// Mitsubishi GX Works2 project: modbus ASCII   PLC: FX1N/FX1NC

PROGRAM MAIN
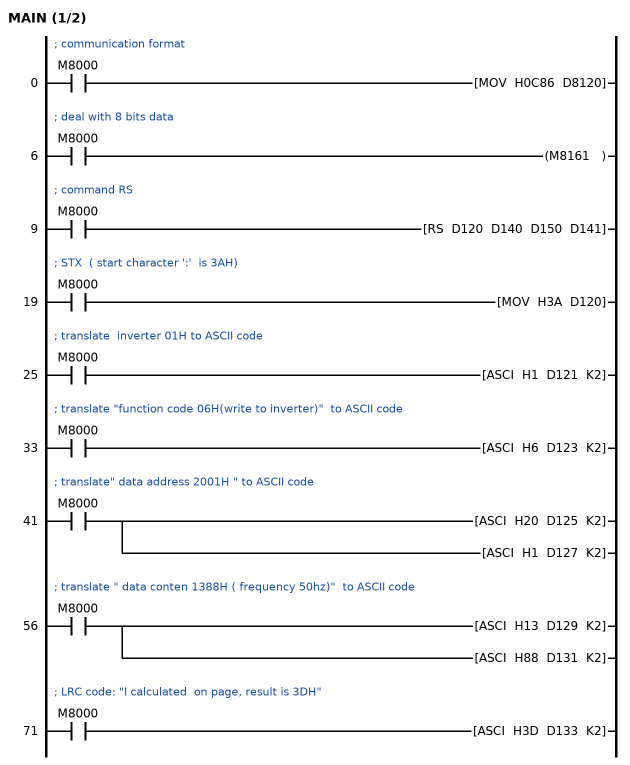
; communication format
0     LD      M8000
      MOV     H0C86 D8120
; deal with 8 bits data
6     LD      M8000
      OUT     M8161
; command RS
9     LD      M8000
      RS      D120 D140 D150 D141
; STX  ( start character ':'  is 3AH)
19    LD      M8000
      MOV     H3A D120
; translate  inverter 01H to ASCII code
25    LD      M8000
      ASCI    H1 D121 K2
; translate "function code 06H(write to inverter)"  to ASCII code
33    LD      M8000
      ASCI    H6 D123 K2
; translate" data address 2001H " to ASCII code
41    LD      M8000
      ASCI    H20 D125 K2
      ASCI    H1 D127 K2
; translate " data conten 1388H ( frequency 50hz)"  to ASCII code
56    LD      M8000
      ASCI    H13 D129 K2
      ASCI    H88 D131 K2
; LRC code: "I calculated  on page, result is 3DH"
71    LD      M8000
      ASCI    H3D D133 K2
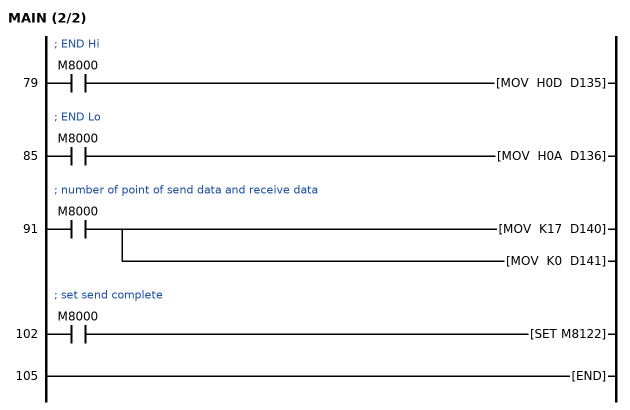
; END Hi
79    LD      M8000
      MOV     H0D D135
; END Lo
85    LD      M8000
      MOV     H0A D136
; number of point of send data and receive data
91    LD      M8000
      MOV     K17 D140
      MOV     K0 D141
; set send complete
102   LD      M8000
      SET     M8122
105   END
END_PROGRAM
